TYPE ST_SlaveArmCtrlCmds :
STRUCT
	// arm control data
	m_jntEnableFlag : Vec8i;
	m_jntOPMode : Vec8i;
	m_cmdJntPos : VEC8d;
	m_cmdJntVel : VEC8d;
	m_cmdJntAcc : VEC8d;
	m_cmdJntTrq : VEC8d;
	m_cmdCartPose : ST_Frame;
	m_cmdCartTwist : Vec6d;
	m_ratedCur : VEC8d;
	
END_STRUCT
END_TYPE

(* stored: Version 1.1.0.1, ProductVersion 3.1.4024.11
   DUT ST_SlaveArmCtrlCmds: Id {0454013e-c8cb-47dd-933d-f5a976121303} *)
